FUNCTION_BLOCK RepairConsumer (* Simple FB with one algorithm *)
  (* Standard: 61499-1 *)
  (* Version 1.0, 2026-07-21, Dimitrios Kalligaridis *)
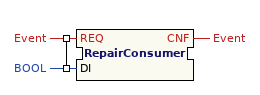
  EVENT_INPUT
    REQ WITH DI; (* Normal Execution Request *)
  END_EVENT
  EVENT_OUTPUT
    CNF; (* Execution Confirmation *)
  END_EVENT
  VAR_INPUT
    DI : BOOL;
  END_VAR
  EC_STATES
    REQ : REQ -> CNF;
  END_STATES
  ALGORITHM REQ IN ST:

  END_ALGORITHM
END_FUNCTION_BLOCK
